// TIA Portal V18 export
FUNCTION_BLOCK "ST10_Flow28_LUnloadingLoad&Unload"   // FB1098, GRAPH
VERSION : 0.1
// stored: AcknowledgeErrorsRequired false, AutoNumber false, GraphVersion 6.0, InitialValuesAcquisition false, IsIECCheckEnabled false, LanguageInNetworks LAD, LockOperatingMode false, PermanentILProcessingInMANMode false, SetENOAutomatically false, SkipSteps false, UDAEnableTagReadback false, WithAlarmHandling true
   // inherited from GRAPH_BASE
   VAR
      OFF_SQ_BASE : Bool;
   END_VAR
   VAR_INPUT
      iSysInface : "RCS_SysComInterface_V1";
   END_VAR
   VAR_IN_OUT
      ioPM_Inface : "RCS_PMInterface_V1";
      ioStatus : Int;
   END_VAR
   VAR
      sCtrlMode { S7_SetPoint := 'True'} : "SysFlowCtrlGraph";
      sUpdMES_Data : Bool;   // 更新MES数据
      工件放行中 : Bool;
      前站站号 { ExternalAccessible := 'False'; ExternalVisible := 'False'; ExternalWritable := 'False'} : UInt;
      本站站号 { ExternalAccessible := 'False'; ExternalVisible := 'False'; ExternalWritable := 'False'} : UInt;
      弹窗Temp : Array[1..10] of Int;
      AlarmID : Int;
      TON { S7_SetPoint := 'True'} : Array[0..10] of TON_TIME;
      TOF { S7_SetPoint := 'True'} : Array[0..10] of TOF_TIME;
      sUP { S7_SetPoint := 'True'} : Array[0..10] of Bool;
      更新RFID完成 : Bool;
   END_VAR
   VAR_TEMP
      Tempresult : USInt;
      本站站号乘10 : UInt;
   END_VAR
   // // TON[0] : 托盘流入1托盘到位传感器 / iA-Rotating product Check
   // // TON[1] : 托盘流入1托盘到位传感器
   // // TON[2] : 托盘流入1产品有无传感器
   // // TON[3] : 托盘流入1产品有无传感器
   // // TON[4] : 托盘流入1姿态检测光电2
   // // TON[5] : 托盘流入1姿态检测光电3
   // // TON[0].Q : 托盘流入1托盘到位 / iA-Rotating product Check
   // // TON[1].Q : 托盘流入1托盘无
   // // TON[2].Q : 托盘流入1有产品
   // // TON[3].Q : 托盘流入1无产品
   // // TON[4].Q : 托盘流入1姿态检测光电2
   // // TON[5].Q : 托盘流入1姿态检测光电3
   // // TOF[1] : iA-Rotating product Check
BEGIN
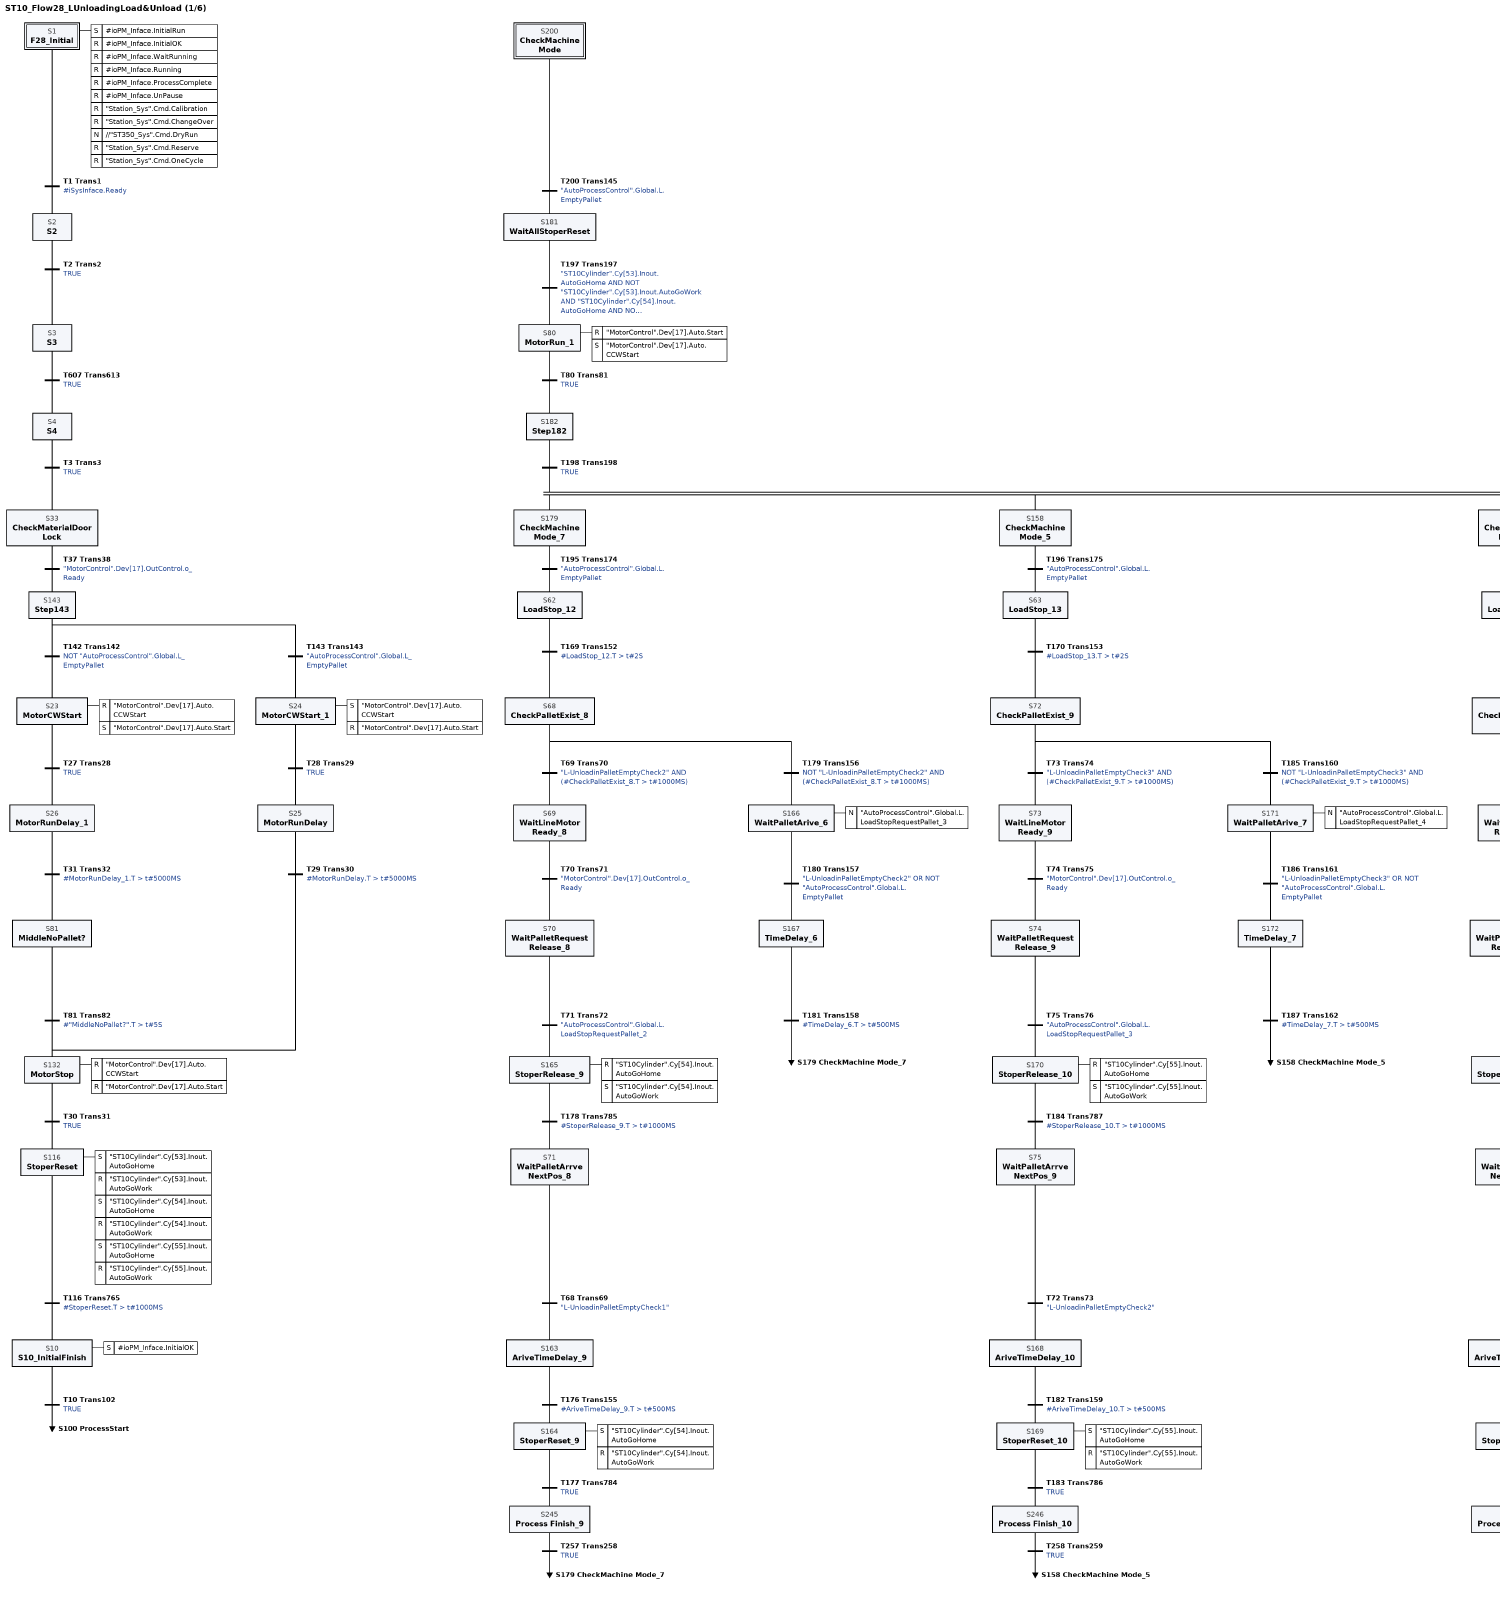
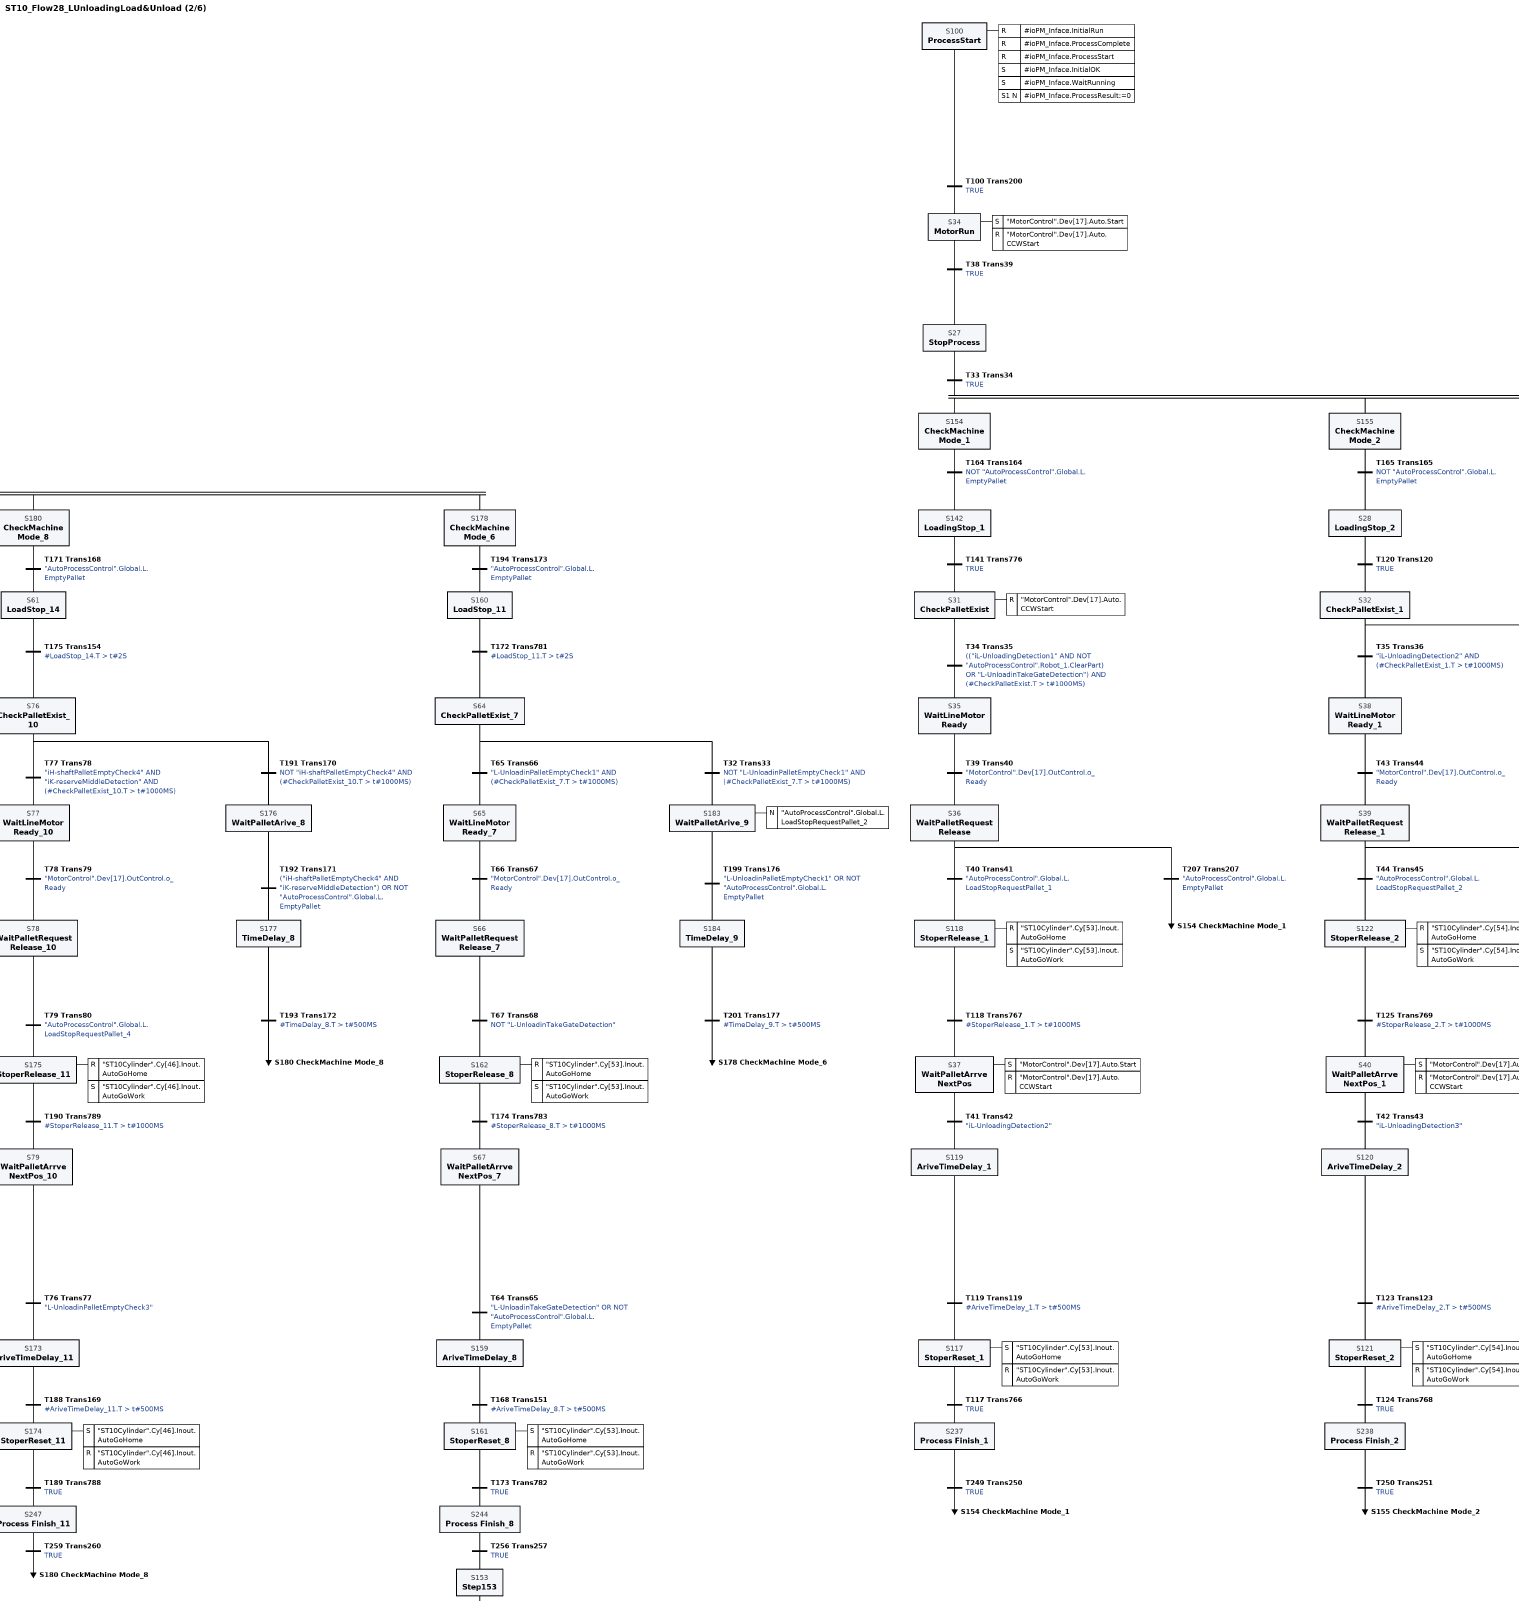
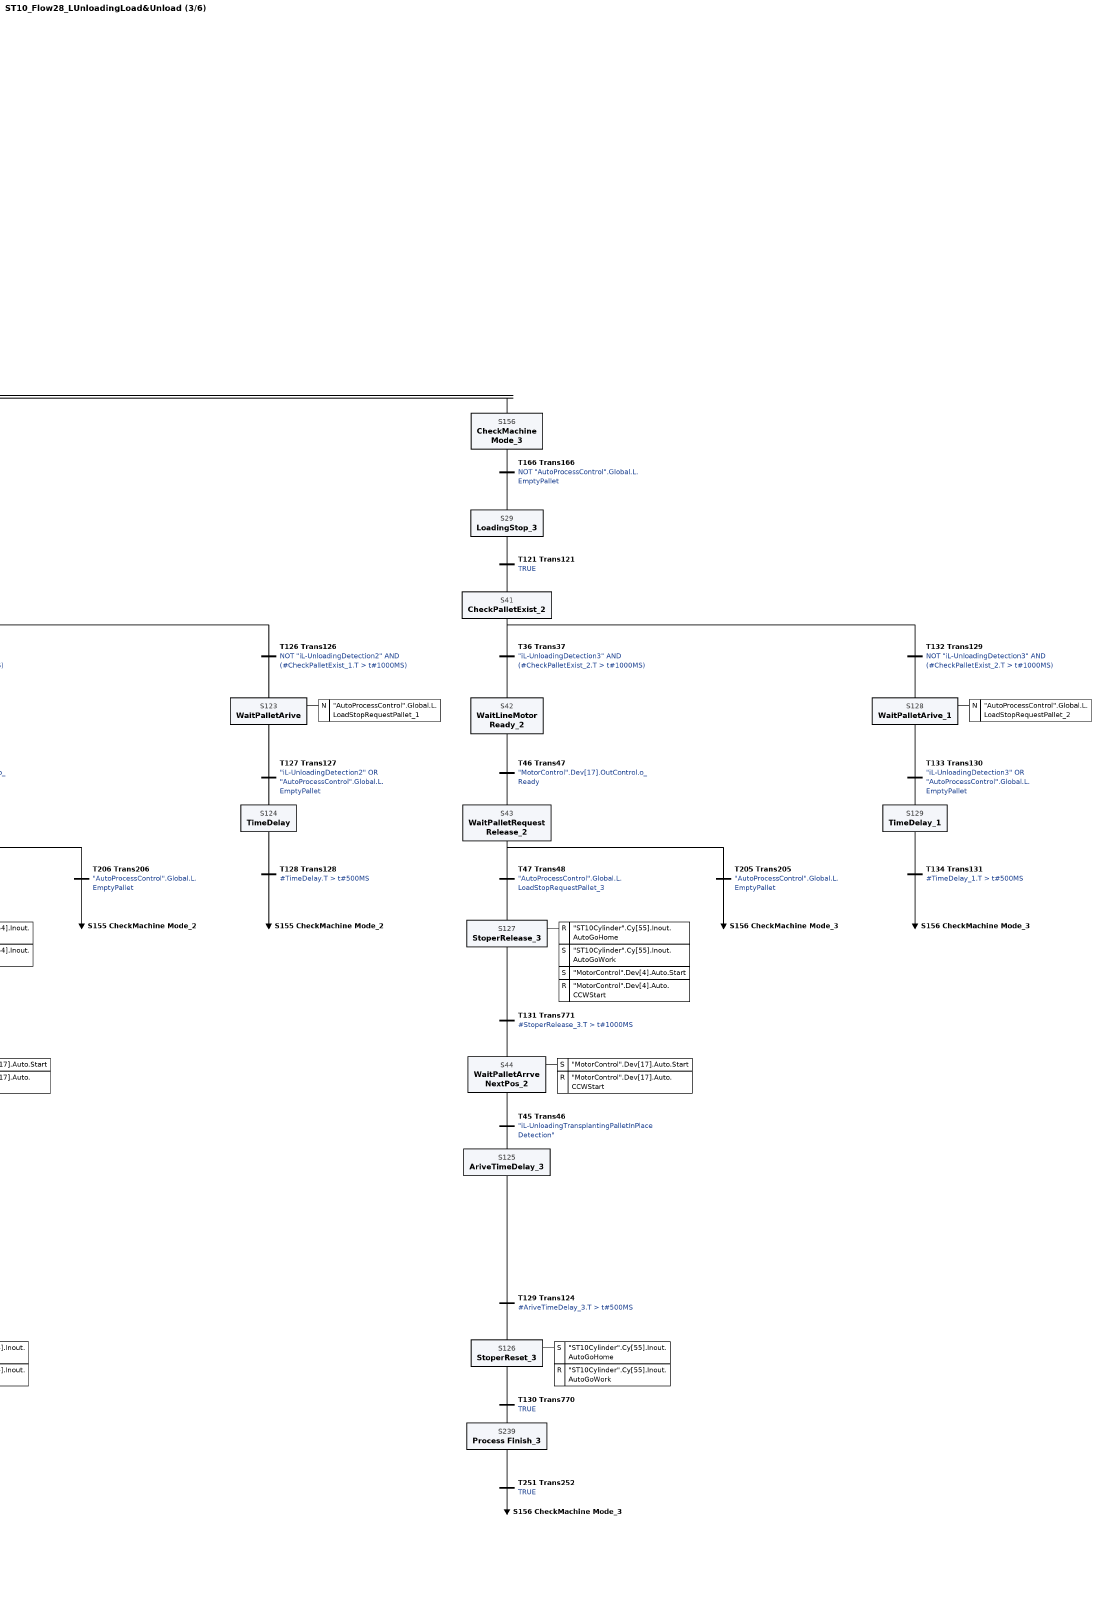
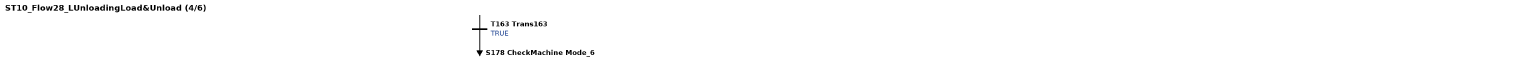
   // permanent pre-instructions
   NETWORK 1
      #TON[10].TON(IN := "AlwaysTRUE" AND "Station_Sys".Alarm.ImmediatelyStop, PT := T#300ms);
      #ioPM_Inface.AlarmImdilyStop := #TON[10].Q;
      #ioPM_Inface.AlarmCycleStop := "AlwaysTRUE" AND "Station_Sys".Alarm.CycleStop;
   NETWORK 2
      IF NOT False THEN
          #sCtrlMode(iSysInface := #iSysInface, ioPM_Inface := #ioPM_Inface, ioGraphCtrl := #RT_DATA.MOP);   // "SysFlowCtrlGraph"
      END_IF;
   NETWORK 3
      #TON[0].TON(IN := "AlwaysTRUE" AND "iK-reserveLifting3PalletDischargeDetection", PT := t#2000ms);   // 工位11有托盘
      #TOF[1].TOF(IN := "AlwaysTRUE" AND NOT "iK-reserveLifting3PalletDischargeDetection", PT := T#300ms);   // 工位无托盘
      #TON[2].TON(IN := "AlwaysTRUE", PT := T#300ms);
      #TOF[3].TOF(IN := "AlwaysTRUE", PT := T#300ms);
      #TON[4].TON(IN := "AlwaysTRUE", PT := T#300ms);
      #TOF[5].TOF(IN := "AlwaysTRUE", PT := T#300ms);
   NETWORK 4
      #前站站号 := 345;
      #本站站号 := 350;

   // sequencer 1: S01-S99 初始化 / S01-S99 Initial
   INITIAL_STEP F28_Initial:   // S1, max time T#10S, warning time T#7S
              S    #ioPM_Inface.InitialRun
              R    #ioPM_Inface.InitialOK
              R    #ioPM_Inface.WaitRunning
              R    #ioPM_Inface.Running
              R    #ioPM_Inface.ProcessComplete
              R    #ioPM_Inface.UnPause
              R    "Station_Sys".Cmd.Calibration
              R    "Station_Sys".Cmd.ChangeOver
                   //"ST350_Sys".Cmd.DryRun
              R    "Station_Sys".Cmd.Reserve
              R    "Station_Sys".Cmd.OneCycle
   END_STEP
   TRANSITION Trans1 FROM F28_Initial TO S2   // T1
      := #iSysInface.Ready;
   END_TRANSITION
   STEP S2:   // S2, max time T#10S, warning time T#7S
   END_STEP
   TRANSITION Trans2 FROM S2 TO S3   // T2
      := TRUE;
   END_TRANSITION
   STEP S4:   // S4, max time T#10S, warning time T#7S
   END_STEP
   TRANSITION Trans3 FROM S4 TO CheckMaterialDoorLock   // T3
      := TRUE;
   END_TRANSITION
   STEP MotorRunDelay_1:   // S26, max time T#10S, warning time T#7S
   END_STEP
   TRANSITION Trans32 FROM MotorRunDelay_1 TO "MiddleNoPallet?"   // T31
      := #MotorRunDelay_1.T > t#5000MS;
   END_TRANSITION
   STEP S10_InitialFinish:   // S10, max time T#10S, warning time T#7S
              S    #ioPM_Inface.InitialOK
   END_STEP
   TRANSITION Trans102 FROM S10_InitialFinish TO ProcessStart   // T10, jump
      := TRUE;
   END_TRANSITION
   STEP S3:   // S3, max time T#10S, warning time T#7S
   END_STEP
   TRANSITION Trans613 FROM S3 TO S4   // T607
      := TRUE;
   END_TRANSITION
   STEP CheckMaterialDoorLock:   // S33, max time T#10S, warning time T#7S
   END_STEP
   TRANSITION Trans38 FROM CheckMaterialDoorLock TO Step143   // T37
      := "MotorControl".Dev[17].OutControl.o_Ready;
   END_TRANSITION
   STEP "MiddleNoPallet?":   // S81, max time T#10S, warning time T#7S
   END_STEP
   TRANSITION Trans82 FROM "MiddleNoPallet?" TO MotorStop   // T81
      := #"MiddleNoPallet?".T > t#5S;
   END_TRANSITION
   STEP StoperReset:   // S116, max time T#10S, warning time T#7S
              S    "ST10Cylinder".Cy[53].Inout.AutoGoHome
              R    "ST10Cylinder".Cy[53].Inout.AutoGoWork
              S    "ST10Cylinder".Cy[54].Inout.AutoGoHome
              R    "ST10Cylinder".Cy[54].Inout.AutoGoWork
              S    "ST10Cylinder".Cy[55].Inout.AutoGoHome
              R    "ST10Cylinder".Cy[55].Inout.AutoGoWork
   END_STEP
   TRANSITION Trans765 FROM StoperReset TO S10_InitialFinish   // T116
      := #StoperReset.T > t#1000MS;
   END_TRANSITION
   STEP MotorCWStart_1:   // S24, max time T#10S, warning time T#7S
              S    "MotorControl".Dev[17].Auto.CCWStart
              R    "MotorControl".Dev[17].Auto.Start
   END_STEP
   TRANSITION Trans29 FROM MotorCWStart_1 TO MotorRunDelay   // T28
      := TRUE;
   END_TRANSITION
   STEP Step143:   // S143, max time T#10S, warning time T#7S
   END_STEP
   TRANSITION Trans142 FROM Step143 TO MotorCWStart   // T142
      := NOT "AutoProcessControl".Global.L_EmptyPallet;
   END_TRANSITION
   TRANSITION Trans143 FROM Step143 TO MotorCWStart_1   // T143
      := "AutoProcessControl".Global.L_EmptyPallet;
   END_TRANSITION
   STEP MotorCWStart:   // S23, max time T#10S, warning time T#7S
              R    "MotorControl".Dev[17].Auto.CCWStart
              S    "MotorControl".Dev[17].Auto.Start
   END_STEP
   TRANSITION Trans28 FROM MotorCWStart TO MotorRunDelay_1   // T27
      := TRUE;
   END_TRANSITION
   STEP MotorStop:   // S132, max time T#10S, warning time T#7S
              R    "MotorControl".Dev[17].Auto.CCWStart
              R    "MotorControl".Dev[17].Auto.Start
   END_STEP
   TRANSITION Trans31 FROM MotorStop TO StoperReset   // T30
      := TRUE;
   END_TRANSITION
   STEP MotorRunDelay:   // S25, max time T#10S, warning time T#7S
   END_STEP
   TRANSITION Trans30 FROM MotorRunDelay TO MotorStop   // T29
      := #MotorRunDelay.T > t#5000MS;
   END_TRANSITION

   // sequencer 2: S100-S199 等待到位 / S100-S199 CheckLineMode
   STEP ProcessStart:   // S100, max time T#10S, warning time T#7S
      // 自动等待开始运行
              R    #ioPM_Inface.InitialRun
              R    #ioPM_Inface.ProcessComplete
              R    #ioPM_Inface.ProcessStart
              S    #ioPM_Inface.InitialOK
              S    #ioPM_Inface.WaitRunning
          S1  N    #ioPM_Inface.ProcessResult:=0
   END_STEP
   TRANSITION Trans200 FROM ProcessStart TO MotorRun   // T100
      := TRUE;
   END_TRANSITION
   STEP "Process Finish_1":   // S237, max time T#10S, warning time T#7S
   END_STEP
   TRANSITION Trans250 FROM "Process Finish_1" TO "CheckMachine Mode_1"   // T249, jump
      := TRUE;
   END_TRANSITION
   STEP StopProcess:   // S27, max time T#10S, warning time T#7S
   END_STEP
   TRANSITION Trans34 FROM StopProcess TO ("CheckMachine Mode_1", "CheckMachine Mode_2", "CheckMachine Mode_3")   // T33
      := TRUE;
   END_TRANSITION
   STEP MotorRun:   // S34, max time T#10S, warning time T#7S
              S    "MotorControl".Dev[17].Auto.Start
              R    "MotorControl".Dev[17].Auto.CCWStart
   END_STEP
   TRANSITION Trans39 FROM MotorRun TO StopProcess   // T38
      := TRUE;
   END_TRANSITION
   STEP LoadingStop_2:   // S28, max time T#10S, warning time T#7S
   END_STEP
   TRANSITION Trans120 FROM LoadingStop_2 TO CheckPalletExist_1   // T120
      := TRUE;
   END_TRANSITION
   STEP "CheckMachine Mode_3":   // S156, max time T#10S, warning time T#7S
   END_STEP
   TRANSITION Trans166 FROM "CheckMachine Mode_3" TO LoadingStop_3   // T166
      := NOT "AutoProcessControl".Global.L.EmptyPallet;
   END_TRANSITION
   STEP LoadingStop_3:   // S29, max time T#10S, warning time T#7S
   END_STEP
   TRANSITION Trans121 FROM LoadingStop_3 TO CheckPalletExist_2   // T121
      := TRUE;
   END_TRANSITION
   STEP CheckPalletExist:   // S31, max time T#10S, warning time T#7S
              R    "MotorControl".Dev[17].Auto.CCWStart
   END_STEP
   TRANSITION Trans35 FROM CheckPalletExist TO WaitLineMotorReady   // T34
      := (("iL-UnloadingDetection1" AND NOT "AutoProcessControl".Robot_1.ClearPart) OR "L-UnloadinTakeGateDetection") AND (#CheckPalletExist.T > t#1000MS);
   END_TRANSITION
   STEP AriveTimeDelay_1:   // S119, max time T#10S, warning time T#7S
   END_STEP
   TRANSITION Trans119 FROM AriveTimeDelay_1 TO StoperReset_1   // T119
      := #AriveTimeDelay_1.T > t#500MS;
   END_TRANSITION
   STEP WaitLineMotorReady:   // S35, max time T#10S, warning time T#7S
   END_STEP
   TRANSITION Trans40 FROM WaitLineMotorReady TO WaitPalletRequestRelease   // T39
      := "MotorControl".Dev[17].OutControl.o_Ready;
   END_TRANSITION
   STEP WaitPalletRequestRelease:   // S36, max time T#10S, warning time T#7S
   END_STEP
   TRANSITION Trans41 FROM WaitPalletRequestRelease TO StoperRelease_1   // T40
      := "AutoProcessControl".Global.L.LoadStopRequestPallet_1;
   END_TRANSITION
   TRANSITION Trans207 FROM WaitPalletRequestRelease TO "CheckMachine Mode_1"   // T207, jump
      := "AutoProcessControl".Global.L.EmptyPallet;
   END_TRANSITION
   STEP LoadingStop_1:   // S142, max time T#10S, warning time T#7S
   END_STEP
   TRANSITION Trans776 FROM LoadingStop_1 TO CheckPalletExist   // T141
      := TRUE;
   END_TRANSITION
   STEP WaitPalletArrveNextPos:   // S37, max time T#10S, warning time T#7S
              S    "MotorControl".Dev[17].Auto.Start
              R    "MotorControl".Dev[17].Auto.CCWStart
   END_STEP
   TRANSITION Trans42 FROM WaitPalletArrveNextPos TO AriveTimeDelay_1   // T41
      := "iL-UnloadingDetection2";
   END_TRANSITION
   STEP "Process Finish_2":   // S238, max time T#10S, warning time T#7S
   END_STEP
   TRANSITION Trans251 FROM "Process Finish_2" TO "CheckMachine Mode_2"   // T250, jump
      := TRUE;
   END_TRANSITION
   STEP StoperReset_1:   // S117, max time T#10S, warning time T#7S
              S    "ST10Cylinder".Cy[53].Inout.AutoGoHome
              R    "ST10Cylinder".Cy[53].Inout.AutoGoWork
   END_STEP
   TRANSITION Trans766 FROM StoperReset_1 TO "Process Finish_1"   // T117
      := TRUE;
   END_TRANSITION
   STEP StoperRelease_1:   // S118, max time T#10S, warning time T#7S
              R    "ST10Cylinder".Cy[53].Inout.AutoGoHome
              S    "ST10Cylinder".Cy[53].Inout.AutoGoWork
   END_STEP
   TRANSITION Trans767 FROM StoperRelease_1 TO WaitPalletArrveNextPos   // T118
      := #StoperRelease_1.T > t#1000MS;
   END_TRANSITION
   STEP CheckPalletExist_1:   // S32, max time T#10S, warning time T#7S
   END_STEP
   TRANSITION Trans36 FROM CheckPalletExist_1 TO WaitLineMotorReady_1   // T35
      := "iL-UnloadingDetection2" AND (#CheckPalletExist_1.T > t#1000MS);
   END_TRANSITION
   TRANSITION Trans126 FROM CheckPalletExist_1 TO WaitPalletArive   // T126
      := NOT "iL-UnloadingDetection2" AND (#CheckPalletExist_1.T > t#1000MS);
   END_TRANSITION
   STEP AriveTimeDelay_2:   // S120, max time T#10S, warning time T#7S
   END_STEP
   TRANSITION Trans123 FROM AriveTimeDelay_2 TO StoperReset_2   // T123
      := #AriveTimeDelay_2.T > t#500MS;
   END_TRANSITION
   STEP WaitLineMotorReady_1:   // S38, max time T#10S, warning time T#7S
   END_STEP
   TRANSITION Trans44 FROM WaitLineMotorReady_1 TO WaitPalletRequestRelease_1   // T43
      := "MotorControl".Dev[17].OutControl.o_Ready;
   END_TRANSITION
   STEP WaitPalletRequestRelease_1:   // S39, max time T#10S, warning time T#7S
   END_STEP
   TRANSITION Trans45 FROM WaitPalletRequestRelease_1 TO StoperRelease_2   // T44
      := "AutoProcessControl".Global.L.LoadStopRequestPallet_2;
   END_TRANSITION
   TRANSITION Trans206 FROM WaitPalletRequestRelease_1 TO "CheckMachine Mode_2"   // T206, jump
      := "AutoProcessControl".Global.L.EmptyPallet;
   END_TRANSITION
   STEP WaitPalletArrveNextPos_1:   // S40, max time T#10S, warning time T#7S
              S    "MotorControl".Dev[17].Auto.Start
              R    "MotorControl".Dev[17].Auto.CCWStart
   END_STEP
   TRANSITION Trans43 FROM WaitPalletArrveNextPos_1 TO AriveTimeDelay_2   // T42
      := "iL-UnloadingDetection3";
   END_TRANSITION
   STEP StoperReset_2:   // S121, max time T#10S, warning time T#7S
              S    "ST10Cylinder".Cy[54].Inout.AutoGoHome
              R    "ST10Cylinder".Cy[54].Inout.AutoGoWork
   END_STEP
   TRANSITION Trans768 FROM StoperReset_2 TO "Process Finish_2"   // T124
      := TRUE;
   END_TRANSITION
   STEP StoperRelease_2:   // S122, max time T#10S, warning time T#7S
              R    "ST10Cylinder".Cy[54].Inout.AutoGoHome
              S    "ST10Cylinder".Cy[54].Inout.AutoGoWork
   END_STEP
   TRANSITION Trans769 FROM StoperRelease_2 TO WaitPalletArrveNextPos_1   // T125
      := #StoperRelease_2.T > t#1000MS;
   END_TRANSITION
   STEP WaitPalletArive:   // S123, max time T#10S, warning time T#7S
              N    "AutoProcessControl".Global.L.LoadStopRequestPallet_1
   END_STEP
   TRANSITION Trans127 FROM WaitPalletArive TO TimeDelay   // T127
      := "iL-UnloadingDetection2" OR "AutoProcessControl".Global.L.EmptyPallet;
   END_TRANSITION
   STEP TimeDelay:   // S124, max time T#10S, warning time T#7S
   END_STEP
   TRANSITION Trans128 FROM TimeDelay TO "CheckMachine Mode_2"   // T128, jump
      := #TimeDelay.T > t#500MS;
   END_TRANSITION
   STEP "Process Finish_3":   // S239, max time T#10S, warning time T#7S
   END_STEP
   TRANSITION Trans252 FROM "Process Finish_3" TO "CheckMachine Mode_3"   // T251, jump
      := TRUE;
   END_TRANSITION
   STEP CheckPalletExist_2:   // S41, max time T#10S, warning time T#7S
   END_STEP
   TRANSITION Trans37 FROM CheckPalletExist_2 TO WaitLineMotorReady_2   // T36
      := "iL-UnloadingDetection3" AND (#CheckPalletExist_2.T > t#1000MS);
   END_TRANSITION
   TRANSITION Trans129 FROM CheckPalletExist_2 TO WaitPalletArive_1   // T132
      := NOT "iL-UnloadingDetection3" AND (#CheckPalletExist_2.T > t#1000MS);
   END_TRANSITION
   STEP AriveTimeDelay_3:   // S125, max time T#10S, warning time T#7S
   END_STEP
   TRANSITION Trans124 FROM AriveTimeDelay_3 TO StoperReset_3   // T129
      := #AriveTimeDelay_3.T > t#500MS;
   END_TRANSITION
   STEP WaitLineMotorReady_2:   // S42, max time T#10S, warning time T#7S
   END_STEP
   TRANSITION Trans47 FROM WaitLineMotorReady_2 TO WaitPalletRequestRelease_2   // T46
      := "MotorControl".Dev[17].OutControl.o_Ready;
   END_TRANSITION
   STEP WaitPalletRequestRelease_2:   // S43, max time T#10S, warning time T#7S
   END_STEP
   TRANSITION Trans48 FROM WaitPalletRequestRelease_2 TO StoperRelease_3   // T47
      := "AutoProcessControl".Global.L.LoadStopRequestPallet_3;
   END_TRANSITION
   TRANSITION Trans205 FROM WaitPalletRequestRelease_2 TO "CheckMachine Mode_3"   // T205, jump
      := "AutoProcessControl".Global.L.EmptyPallet;
   END_TRANSITION
   STEP WaitPalletArrveNextPos_2:   // S44, max time T#10S, warning time T#7S
              S    "MotorControl".Dev[17].Auto.Start
              R    "MotorControl".Dev[17].Auto.CCWStart
   END_STEP
   TRANSITION Trans46 FROM WaitPalletArrveNextPos_2 TO AriveTimeDelay_3   // T45
      := "iL-UnloadingTransplantingPalletInPlaceDetection";
   END_TRANSITION
   STEP StoperReset_3:   // S126, max time T#10S, warning time T#7S
              S    "ST10Cylinder".Cy[55].Inout.AutoGoHome
              R    "ST10Cylinder".Cy[55].Inout.AutoGoWork
   END_STEP
   TRANSITION Trans770 FROM StoperReset_3 TO "Process Finish_3"   // T130
      := TRUE;
   END_TRANSITION
   STEP StoperRelease_3:   // S127, max time T#10S, warning time T#7S
              R    "ST10Cylinder".Cy[55].Inout.AutoGoHome
              S    "ST10Cylinder".Cy[55].Inout.AutoGoWork
              S    "MotorControl".Dev[4].Auto.Start
              R    "MotorControl".Dev[4].Auto.CCWStart
   END_STEP
   TRANSITION Trans771 FROM StoperRelease_3 TO WaitPalletArrveNextPos_2   // T131
      := #StoperRelease_3.T > t#1000MS;
   END_TRANSITION
   STEP WaitPalletArive_1:   // S128, max time T#10S, warning time T#7S
              N    "AutoProcessControl".Global.L.LoadStopRequestPallet_2
   END_STEP
   TRANSITION Trans130 FROM WaitPalletArive_1 TO TimeDelay_1   // T133
      := "iL-UnloadingDetection3" OR "AutoProcessControl".Global.L.EmptyPallet;
   END_TRANSITION
   STEP TimeDelay_1:   // S129, max time T#10S, warning time T#7S
   END_STEP
   TRANSITION Trans131 FROM TimeDelay_1 TO "CheckMachine Mode_3"   // T134, jump
      := #TimeDelay_1.T > t#500MS;
   END_TRANSITION
   STEP "CheckMachine Mode_1":   // S154, max time T#10S, warning time T#7S
   END_STEP
   TRANSITION Trans164 FROM "CheckMachine Mode_1" TO LoadingStop_1   // T164
      := NOT "AutoProcessControl".Global.L.EmptyPallet;
   END_TRANSITION
   STEP "CheckMachine Mode_2":   // S155, max time T#10S, warning time T#7S
   END_STEP
   TRANSITION Trans165 FROM "CheckMachine Mode_2" TO LoadingStop_2   // T165
      := NOT "AutoProcessControl".Global.L.EmptyPallet;
   END_TRANSITION

   // sequencer 3: Empty Process
   INITIAL_STEP CheckMachineMode:   // S200, max time T#10S, warning time T#7S
   END_STEP
   TRANSITION Trans145 FROM CheckMachineMode TO WaitAllStoperReset   // T200
      := "AutoProcessControl".Global.L.EmptyPallet;
   END_TRANSITION
   STEP Step153:   // S153, max time T#10S, warning time T#7S
   END_STEP
   TRANSITION Trans163 FROM Step153 TO "CheckMachine Mode_6"   // T163, jump
      := TRUE;
   END_TRANSITION
   STEP "Process Finish_8":   // S244, max time T#10S, warning time T#7S
   END_STEP
   TRANSITION Trans257 FROM "Process Finish_8" TO Step153   // T256
      := TRUE;
   END_TRANSITION
   STEP LoadStop_14:   // S61, max time T#10S, warning time T#7S
   END_STEP
   TRANSITION Trans154 FROM LoadStop_14 TO CheckPalletExist_10   // T175
      := #LoadStop_14.T > t#2S;
   END_TRANSITION
   STEP LoadStop_12:   // S62, max time T#10S, warning time T#7S
   END_STEP
   TRANSITION Trans152 FROM LoadStop_12 TO CheckPalletExist_8   // T169
      := #LoadStop_12.T > t#2S;
   END_TRANSITION
   STEP "CheckMachine Mode_5":   // S158, max time T#10S, warning time T#7S
   END_STEP
   TRANSITION Trans175 FROM "CheckMachine Mode_5" TO LoadStop_13   // T196
      := "AutoProcessControl".Global.L.EmptyPallet;
   END_TRANSITION
   STEP LoadStop_13:   // S63, max time T#10S, warning time T#7S
   END_STEP
   TRANSITION Trans153 FROM LoadStop_13 TO CheckPalletExist_9   // T170
      := #LoadStop_13.T > t#2S;
   END_TRANSITION
   STEP CheckPalletExist_7:   // S64, max time T#10S, warning time T#7S
   END_STEP
   TRANSITION Trans66 FROM CheckPalletExist_7 TO WaitLineMotorReady_7   // T65
      := "L-UnloadinPalletEmptyCheck1" AND (#CheckPalletExist_7.T > t#1000MS);
   END_TRANSITION
   TRANSITION Trans33 FROM CheckPalletExist_7 TO WaitPalletArive_9   // T32
      := NOT "L-UnloadinPalletEmptyCheck1" AND (#CheckPalletExist_7.T > t#1000MS);
   END_TRANSITION
   STEP AriveTimeDelay_8:   // S159, max time T#10S, warning time T#7S
   END_STEP
   TRANSITION Trans151 FROM AriveTimeDelay_8 TO StoperReset_8   // T168
      := #AriveTimeDelay_8.T > t#500MS;
   END_TRANSITION
   STEP WaitLineMotorReady_7:   // S65, max time T#10S, warning time T#7S
   END_STEP
   TRANSITION Trans67 FROM WaitLineMotorReady_7 TO WaitPalletRequestRelease_7   // T66
      := "MotorControl".Dev[17].OutControl.o_Ready;
   END_TRANSITION
   STEP WaitPalletRequestRelease_7:   // S66, max time T#10S, warning time T#7S
   END_STEP
   TRANSITION Trans68 FROM WaitPalletRequestRelease_7 TO StoperRelease_8   // T67
      := NOT "L-UnloadinTakeGateDetection";
   END_TRANSITION
   STEP LoadStop_11:   // S160, max time T#10S, warning time T#7S
   END_STEP
   TRANSITION Trans781 FROM LoadStop_11 TO CheckPalletExist_7   // T172
      := #LoadStop_11.T > t#2S;
   END_TRANSITION
   STEP WaitPalletArrveNextPos_7:   // S67, max time T#10S, warning time T#7S
   END_STEP
   TRANSITION Trans65 FROM WaitPalletArrveNextPos_7 TO AriveTimeDelay_8   // T64
      := "L-UnloadinTakeGateDetection" OR NOT "AutoProcessControl".Global.L.EmptyPallet;
   END_TRANSITION
   STEP "Process Finish_9":   // S245, max time T#10S, warning time T#7S
   END_STEP
   TRANSITION Trans258 FROM "Process Finish_9" TO "CheckMachine Mode_7"   // T257, jump
      := TRUE;
   END_TRANSITION
   STEP StoperReset_8:   // S161, max time T#10S, warning time T#7S
              S    "ST10Cylinder".Cy[53].Inout.AutoGoHome
              R    "ST10Cylinder".Cy[53].Inout.AutoGoWork
   END_STEP
   TRANSITION Trans782 FROM StoperReset_8 TO "Process Finish_8"   // T173
      := TRUE;
   END_TRANSITION
   STEP StoperRelease_8:   // S162, max time T#10S, warning time T#7S
              R    "ST10Cylinder".Cy[53].Inout.AutoGoHome
              S    "ST10Cylinder".Cy[53].Inout.AutoGoWork
   END_STEP
   TRANSITION Trans783 FROM StoperRelease_8 TO WaitPalletArrveNextPos_7   // T174
      := #StoperRelease_8.T > t#1000MS;
   END_TRANSITION
   STEP CheckPalletExist_8:   // S68, max time T#10S, warning time T#7S
   END_STEP
   TRANSITION Trans70 FROM CheckPalletExist_8 TO WaitLineMotorReady_8   // T69
      := "L-UnloadinPalletEmptyCheck2" AND (#CheckPalletExist_8.T > t#1000MS);
   END_TRANSITION
   TRANSITION Trans156 FROM CheckPalletExist_8 TO WaitPalletArive_6   // T179
      := NOT "L-UnloadinPalletEmptyCheck2" AND (#CheckPalletExist_8.T > t#1000MS);
   END_TRANSITION
   STEP AriveTimeDelay_9:   // S163, max time T#10S, warning time T#7S
   END_STEP
   TRANSITION Trans155 FROM AriveTimeDelay_9 TO StoperReset_9   // T176
      := #AriveTimeDelay_9.T > t#500MS;
   END_TRANSITION
   STEP WaitLineMotorReady_8:   // S69, max time T#10S, warning time T#7S
   END_STEP
   TRANSITION Trans71 FROM WaitLineMotorReady_8 TO WaitPalletRequestRelease_8   // T70
      := "MotorControl".Dev[17].OutControl.o_Ready;
   END_TRANSITION
   STEP WaitPalletRequestRelease_8:   // S70, max time T#10S, warning time T#7S
   END_STEP
   TRANSITION Trans72 FROM WaitPalletRequestRelease_8 TO StoperRelease_9   // T71
      := "AutoProcessControl".Global.L.LoadStopRequestPallet_2;
   END_TRANSITION
   STEP WaitPalletArrveNextPos_8:   // S71, max time T#10S, warning time T#7S
   END_STEP
   TRANSITION Trans69 FROM WaitPalletArrveNextPos_8 TO AriveTimeDelay_9   // T68
      := "L-UnloadinPalletEmptyCheck1";
   END_TRANSITION
   STEP StoperReset_9:   // S164, max time T#10S, warning time T#7S
              S    "ST10Cylinder".Cy[54].Inout.AutoGoHome
              R    "ST10Cylinder".Cy[54].Inout.AutoGoWork
   END_STEP
   TRANSITION Trans784 FROM StoperReset_9 TO "Process Finish_9"   // T177
      := TRUE;
   END_TRANSITION
   STEP StoperRelease_9:   // S165, max time T#10S, warning time T#7S
              R    "ST10Cylinder".Cy[54].Inout.AutoGoHome
              S    "ST10Cylinder".Cy[54].Inout.AutoGoWork
   END_STEP
   TRANSITION Trans785 FROM StoperRelease_9 TO WaitPalletArrveNextPos_8   // T178
      := #StoperRelease_9.T > t#1000MS;
   END_TRANSITION
   STEP WaitPalletArive_6:   // S166, max time T#10S, warning time T#7S
              N    "AutoProcessControl".Global.L.LoadStopRequestPallet_3
   END_STEP
   TRANSITION Trans157 FROM WaitPalletArive_6 TO TimeDelay_6   // T180
      := "L-UnloadinPalletEmptyCheck2" OR NOT "AutoProcessControl".Global.L.EmptyPallet;
   END_TRANSITION
   STEP TimeDelay_6:   // S167, max time T#10S, warning time T#7S
   END_STEP
   TRANSITION Trans158 FROM TimeDelay_6 TO "CheckMachine Mode_7"   // T181, jump
      := #TimeDelay_6.T > t#500MS;
   END_TRANSITION
   STEP "Process Finish_10":   // S246, max time T#10S, warning time T#7S
   END_STEP
   TRANSITION Trans259 FROM "Process Finish_10" TO "CheckMachine Mode_5"   // T258, jump
      := TRUE;
   END_TRANSITION
   STEP CheckPalletExist_9:   // S72, max time T#10S, warning time T#7S
   END_STEP
   TRANSITION Trans74 FROM CheckPalletExist_9 TO WaitLineMotorReady_9   // T73
      := "L-UnloadinPalletEmptyCheck3" AND (#CheckPalletExist_9.T > t#1000MS);
   END_TRANSITION
   TRANSITION Trans160 FROM CheckPalletExist_9 TO WaitPalletArive_7   // T185
      := NOT "L-UnloadinPalletEmptyCheck3" AND (#CheckPalletExist_9.T > t#1000MS);
   END_TRANSITION
   STEP AriveTimeDelay_10:   // S168, max time T#10S, warning time T#7S
   END_STEP
   TRANSITION Trans159 FROM AriveTimeDelay_10 TO StoperReset_10   // T182
      := #AriveTimeDelay_10.T > t#500MS;
   END_TRANSITION
   STEP WaitLineMotorReady_9:   // S73, max time T#10S, warning time T#7S
   END_STEP
   TRANSITION Trans75 FROM WaitLineMotorReady_9 TO WaitPalletRequestRelease_9   // T74
      := "MotorControl".Dev[17].OutControl.o_Ready;
   END_TRANSITION
   STEP WaitPalletRequestRelease_9:   // S74, max time T#10S, warning time T#7S
   END_STEP
   TRANSITION Trans76 FROM WaitPalletRequestRelease_9 TO StoperRelease_10   // T75
      := "AutoProcessControl".Global.L.LoadStopRequestPallet_3;
   END_TRANSITION
   STEP WaitPalletArrveNextPos_9:   // S75, max time T#10S, warning time T#7S
   END_STEP
   TRANSITION Trans73 FROM WaitPalletArrveNextPos_9 TO AriveTimeDelay_10   // T72
      := "L-UnloadinPalletEmptyCheck2";
   END_TRANSITION
   STEP StoperReset_10:   // S169, max time T#10S, warning time T#7S
              S    "ST10Cylinder".Cy[55].Inout.AutoGoHome
              R    "ST10Cylinder".Cy[55].Inout.AutoGoWork
   END_STEP
   TRANSITION Trans786 FROM StoperReset_10 TO "Process Finish_10"   // T183
      := TRUE;
   END_TRANSITION
   STEP StoperRelease_10:   // S170, max time T#10S, warning time T#7S
              R    "ST10Cylinder".Cy[55].Inout.AutoGoHome
              S    "ST10Cylinder".Cy[55].Inout.AutoGoWork
   END_STEP
   TRANSITION Trans787 FROM StoperRelease_10 TO WaitPalletArrveNextPos_9   // T184
      := #StoperRelease_10.T > t#1000MS;
   END_TRANSITION
   STEP WaitPalletArive_7:   // S171, max time T#10S, warning time T#7S
              N    "AutoProcessControl".Global.L.LoadStopRequestPallet_4
   END_STEP
   TRANSITION Trans161 FROM WaitPalletArive_7 TO TimeDelay_7   // T186
      := "L-UnloadinPalletEmptyCheck3" OR NOT "AutoProcessControl".Global.L.EmptyPallet;
   END_TRANSITION
   STEP TimeDelay_7:   // S172, max time T#10S, warning time T#7S
   END_STEP
   TRANSITION Trans162 FROM TimeDelay_7 TO "CheckMachine Mode_5"   // T187, jump
      := #TimeDelay_7.T > t#500MS;
   END_TRANSITION
   STEP "Process Finish_11":   // S247, max time T#10S, warning time T#7S
   END_STEP
   TRANSITION Trans260 FROM "Process Finish_11" TO "CheckMachine Mode_8"   // T259, jump
      := TRUE;
   END_TRANSITION
   STEP CheckPalletExist_10:   // S76, max time T#10S, warning time T#7S
   END_STEP
   TRANSITION Trans78 FROM CheckPalletExist_10 TO WaitLineMotorReady_10   // T77
      := "iH-shaftPalletEmptyCheck4" AND "iK-reserveMiddleDetection" AND (#CheckPalletExist_10.T > t#1000MS);
   END_TRANSITION
   TRANSITION Trans170 FROM CheckPalletExist_10 TO WaitPalletArive_8   // T191
      := NOT "iH-shaftPalletEmptyCheck4" AND (#CheckPalletExist_10.T > t#1000MS);
   END_TRANSITION
   STEP AriveTimeDelay_11:   // S173, max time T#10S, warning time T#7S
   END_STEP
   TRANSITION Trans169 FROM AriveTimeDelay_11 TO StoperReset_11   // T188
      := #AriveTimeDelay_11.T > t#500MS;
   END_TRANSITION
   STEP WaitLineMotorReady_10:   // S77, max time T#10S, warning time T#7S
   END_STEP
   TRANSITION Trans79 FROM WaitLineMotorReady_10 TO WaitPalletRequestRelease_10   // T78
      := "MotorControl".Dev[17].OutControl.o_Ready;
   END_TRANSITION
   STEP WaitPalletRequestRelease_10:   // S78, max time T#10S, warning time T#7S
   END_STEP
   TRANSITION Trans80 FROM WaitPalletRequestRelease_10 TO StoperRelease_11   // T79
      := "AutoProcessControl".Global.L.LoadStopRequestPallet_4;
   END_TRANSITION
   STEP WaitPalletArrveNextPos_10:   // S79, max time T#10S, warning time T#7S
   END_STEP
   TRANSITION Trans77 FROM WaitPalletArrveNextPos_10 TO AriveTimeDelay_11   // T76
      := "L-UnloadinPalletEmptyCheck3";
   END_TRANSITION
   STEP StoperReset_11:   // S174, max time T#10S, warning time T#7S
              S    "ST10Cylinder".Cy[46].Inout.AutoGoHome
              R    "ST10Cylinder".Cy[46].Inout.AutoGoWork
   END_STEP
   TRANSITION Trans788 FROM StoperReset_11 TO "Process Finish_11"   // T189
      := TRUE;
   END_TRANSITION
   STEP StoperRelease_11:   // S175, max time T#10S, warning time T#7S
              R    "ST10Cylinder".Cy[46].Inout.AutoGoHome
              S    "ST10Cylinder".Cy[46].Inout.AutoGoWork
   END_STEP
   TRANSITION Trans789 FROM StoperRelease_11 TO WaitPalletArrveNextPos_10   // T190
      := #StoperRelease_11.T > t#1000MS;
   END_TRANSITION
   STEP WaitPalletArive_8:   // S176, max time T#10S, warning time T#7S
   END_STEP
   TRANSITION Trans171 FROM WaitPalletArive_8 TO TimeDelay_8   // T192
      := ("iH-shaftPalletEmptyCheck4" AND "iK-reserveMiddleDetection") OR NOT "AutoProcessControl".Global.L.EmptyPallet;
   END_TRANSITION
   STEP TimeDelay_8:   // S177, max time T#10S, warning time T#7S
   END_STEP
   TRANSITION Trans172 FROM TimeDelay_8 TO "CheckMachine Mode_8"   // T193, jump
      := #TimeDelay_8.T > t#500MS;
   END_TRANSITION
   STEP "CheckMachine Mode_6":   // S178, max time T#10S, warning time T#7S
   END_STEP
   TRANSITION Trans173 FROM "CheckMachine Mode_6" TO LoadStop_11   // T194
      := "AutoProcessControl".Global.L.EmptyPallet;
   END_TRANSITION
   STEP "CheckMachine Mode_7":   // S179, max time T#10S, warning time T#7S
   END_STEP
   TRANSITION Trans174 FROM "CheckMachine Mode_7" TO LoadStop_12   // T195
      := "AutoProcessControl".Global.L.EmptyPallet;
   END_TRANSITION
   STEP "CheckMachine Mode_8":   // S180, max time T#10S, warning time T#7S
   END_STEP
   TRANSITION Trans168 FROM "CheckMachine Mode_8" TO LoadStop_14   // T171
      := "AutoProcessControl".Global.L.EmptyPallet;
   END_TRANSITION
   STEP WaitAllStoperReset:   // S181, max time T#10S, warning time T#7S
   END_STEP
   TRANSITION Trans197 FROM WaitAllStoperReset TO MotorRun_1   // T197
      := "ST10Cylinder".Cy[53].Inout.AutoGoHome AND NOT "ST10Cylinder".Cy[53].Inout.AutoGoWork AND "ST10Cylinder".Cy[54].Inout.AutoGoHome AND NOT "ST10Cylinder".Cy[54].Inout.AutoGoWork AND "ST10Cylinder".Cy[55].Inout.AutoGoHome AND NOT "ST10Cylinder".Cy[55].Inout.AutoGoWork;
   END_TRANSITION
   STEP Step182:   // S182, max time T#10S, warning time T#7S
   END_STEP
   TRANSITION Trans198 FROM Step182 TO ("CheckMachine Mode_7", "CheckMachine Mode_5", "CheckMachine Mode_8", "CheckMachine Mode_6")   // T198
      := TRUE;
   END_TRANSITION
   STEP MotorRun_1:   // S80, max time T#10S, warning time T#7S
              R    "MotorControl".Dev[17].Auto.Start
              S    "MotorControl".Dev[17].Auto.CCWStart
   END_STEP
   TRANSITION Trans81 FROM MotorRun_1 TO Step182   // T80
      := TRUE;
   END_TRANSITION
   STEP WaitPalletArive_9:   // S183, max time T#10S, warning time T#7S
              N    "AutoProcessControl".Global.L.LoadStopRequestPallet_2
   END_STEP
   TRANSITION Trans176 FROM WaitPalletArive_9 TO TimeDelay_9   // T199
      := "L-UnloadinPalletEmptyCheck1" OR NOT "AutoProcessControl".Global.L.EmptyPallet;
   END_TRANSITION
   STEP TimeDelay_9:   // S184, max time T#10S, warning time T#7S
   END_STEP
   TRANSITION Trans177 FROM TimeDelay_9 TO "CheckMachine Mode_6"   // T201, jump
      := #TimeDelay_9.T > t#500MS;
   END_TRANSITION

   // permanent post-instructions
   NETWORK 1
      #ioPM_Inface.StepNum := #RT_DATA.S_DISPLAY;
   NETWORK 2
      IF #iSysInface.Reset THEN #AlarmID := 0; END_IF;
   NETWORK 3
      #TON[10].TON(IN := #工件放行中, PT := T#0.5S);
      IF #TON[10].Q THEN #工件放行中 := FALSE; END_IF;
END_FUNCTION_BLOCK
